// TIA Portal project "template" (V15)

(* hardware
DEVICE "S7-1200 station_1"  S7-1200 Station
   slot 0: "Rack_0"  S7-1200 Rack  Rack  V1.0
   slot 1: "PLC_1"  CPU 1214C AC/DC/Rly  6ES7 214-1BG40-0XB0  V4.2
*)

// ===== PLC "PLC_1"  CPU 1214C AC/DC/Rly =====

VAR_GLOBAL   // PLC tag table "默认变量表"
   "M4.0" AT %M4.0 : Bool;
   "on/off" AT %I0.7 : Bool;
   "start" AT %I0.0 : Bool;
   "M4.1" AT %M4.1 : Bool;
   "water full" AT %I0.1 : Bool;
   "M4.2" AT %M4.2 : Bool;
   "M4.3" AT %M4.3 : Bool;
   "M4.4" AT %M4.4 : Bool;
   "M4.5" AT %M4.5 : Bool;
   "M4.6" AT %M4.6 : Bool;
   "M4.7" AT %M4.7 : Bool;
   "M5.0" AT %M5.0 : Bool;
   "M5.1" AT %M5.1 : Bool;
   "M5.2" AT %M5.2 : Bool;
   "?????????????????" AT %IW30 : Word;
   "cycle of span" AT %MB30 : Byte;
   "cycle of step" AT %MB31 : Byte;
   "water on" AT %Q0.0 : Bool;
   "run+" AT %Q0.1 : Bool;
   "run-" AT %Q0.2 : Bool;
   "tag1" AT %M0.5 : Bool;
   "water off" AT %Q0.3 : Bool;
   "tag2" AT %M0.6 : Bool;
   "water fuck" AT %Q0.4 : Bool;
   "ring" AT %Q0.5 : Bool;
   "stop!!!" AT %I0.2 : Bool;
   "water out" AT %I0.3 : Bool;
   "spanreset" AT %M0.7 : Bool;
   "stepreset" AT %M0.4 : Bool;
END_VAR

// folder: System blocks/Program resources

DATA_BLOCK "IEC_Timer_0_DB"   // DB1
{ S7_Optimized_Access := 'TRUE' }
AUTHOR : Simatic
FAMILY : IEC
NAME : IEC_TMR
VERSION : 1.0
// stored: InstanceOfName IEC_TIMER
"IEC_TIMER"
BEGIN
END_DATA_BLOCK

DATA_BLOCK "IEC_Timer_0_DB_1"   // DB2
{ S7_Optimized_Access := 'TRUE' }
AUTHOR : Simatic
FAMILY : IEC
NAME : IEC_TMR
VERSION : 1.0
// stored: InstanceOfName IEC_TIMER
"IEC_TIMER"
BEGIN
END_DATA_BLOCK

DATA_BLOCK "IEC_Timer_0_DB_2"   // DB3
{ S7_Optimized_Access := 'TRUE' }
AUTHOR : Simatic
FAMILY : IEC
NAME : IEC_TMR
VERSION : 1.0
// stored: InstanceOfName IEC_TIMER
"IEC_TIMER"
BEGIN
END_DATA_BLOCK

DATA_BLOCK "IEC_Timer_0_DB_3"   // DB4
{ S7_Optimized_Access := 'TRUE' }
AUTHOR : Simatic
FAMILY : IEC
NAME : IEC_TMR
VERSION : 1.0
// stored: InstanceOfName IEC_TIMER
"IEC_TIMER"
BEGIN
END_DATA_BLOCK

DATA_BLOCK "IEC_Timer_0_DB_4"   // DB5
{ S7_Optimized_Access := 'TRUE' }
AUTHOR : Simatic
FAMILY : IEC
NAME : IEC_TMR
VERSION : 1.0
// stored: InstanceOfName IEC_TIMER
"IEC_TIMER"
BEGIN
END_DATA_BLOCK

DATA_BLOCK "IEC_Timer_0_DB_5"   // DB6
{ S7_Optimized_Access := 'TRUE' }
AUTHOR : Simatic
FAMILY : IEC
NAME : IEC_TMR
VERSION : 1.0
// stored: InstanceOfName IEC_TIMER
"IEC_TIMER"
BEGIN
END_DATA_BLOCK

DATA_BLOCK "IEC_Timer_0_DB_6"   // DB7
{ S7_Optimized_Access := 'TRUE' }
AUTHOR : Simatic
FAMILY : IEC
NAME : IEC_TMR
VERSION : 1.0
// stored: InstanceOfName IEC_TIMER
"IEC_TIMER"
BEGIN
END_DATA_BLOCK

DATA_BLOCK "IEC_Counter_0_DB"   // DB8
{ S7_Optimized_Access := 'TRUE' }
AUTHOR : Simatic
FAMILY : IEC
NAME : CNTR
VERSION : 1.0
// stored: InstanceOfName IEC_COUNTER
"IEC_COUNTER"
BEGIN
END_DATA_BLOCK

DATA_BLOCK "IEC_Counter_0_DB_1"   // DB9
{ S7_Optimized_Access := 'TRUE' }
AUTHOR : Simatic
FAMILY : IEC
NAME : CNTR
VERSION : 1.0
// stored: InstanceOfName IEC_COUNTER
"IEC_COUNTER"
BEGIN
END_DATA_BLOCK

// folder: (top level)

FUNCTION "STOP" : Void   // FC1, LAD
{ S7_Optimized_Access := 'TRUE' }
VERSION : 0.1
   VAR_INPUT
      "STEP" : Bool;
   END_VAR
BEGIN

REGION Network 1
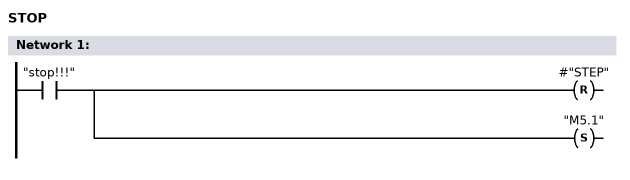
   RUNG wire#powerrail
      Contact( "stop!!!" )
      wire#w1
      R_Coil( #"STEP" )
   END_RUNG
   RUNG wire#w1
      S_Coil( "M5.1" )
   END_RUNG
   // the same network as SCL:
   IF "stop!!!" THEN
       #"STEP" := FALSE;
       "M5.1" := TRUE;
   END_IF;
END_REGION
END_FUNCTION

ORGANIZATION_BLOCK "Main"   // OB1, LAD, ProgramCycle
TITLE = "Main Program Sweep (Cycle)"
{ S7_Optimized_Access := 'TRUE' }
VERSION : 0.1
   VAR_INPUT
      Initial_Call : Bool;   // Initial call of this OB
      Remanence : Bool;   // =True, if remanent data are available
   END_VAR
   VAR_TEMP   // added for the SCL form of the ladder/FBD networks
      _w1 : Bool;
      _w2 : Bool;
      _w3 : Bool;
      _w4 : Bool;
      _w5 : Bool;
      _w6 : Bool;
      _w7 : Bool;
      _w8 : Bool;
      _w9 : Bool;
      _w10 : Bool;
      _w11 : Bool;
      _w12 : Bool;
      _w13 : Bool;
      _w14 : Bool;
      _w15 : Bool;
      _w16 : Bool;
      _w17 : Bool;
      _w18 : Bool;
      _w19 : Bool;
      _w20 : Bool;
   END_VAR
BEGIN

REGION Network 1
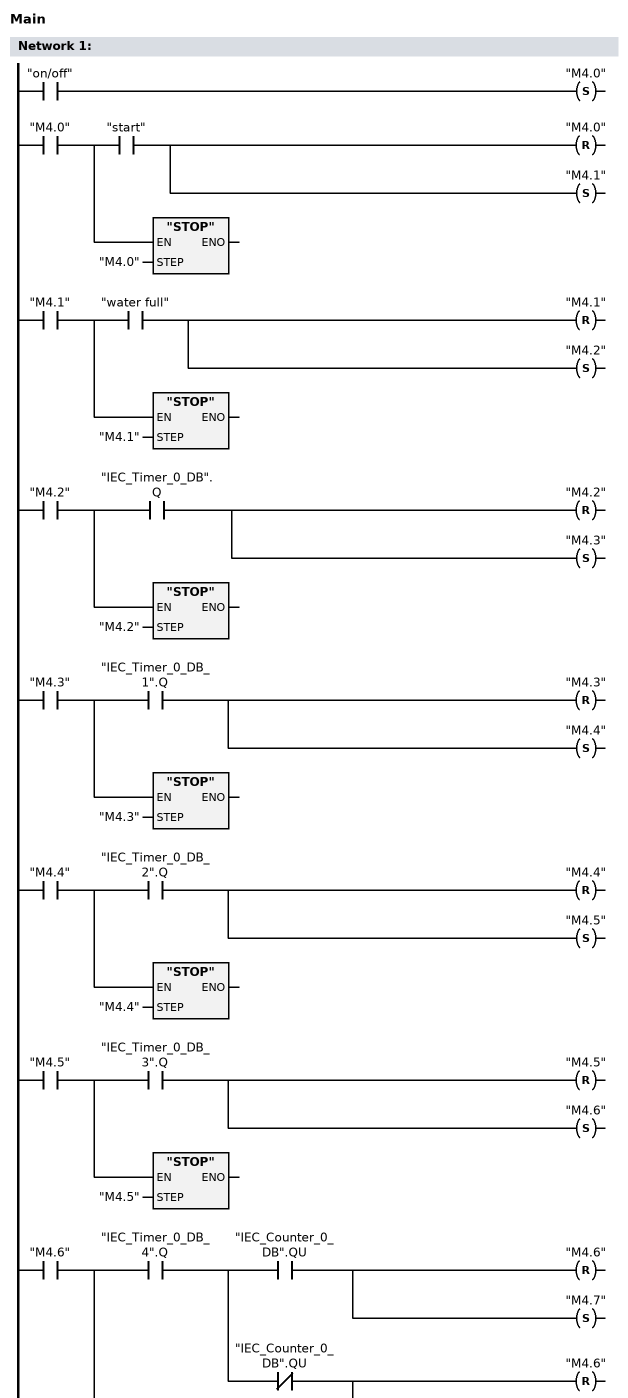
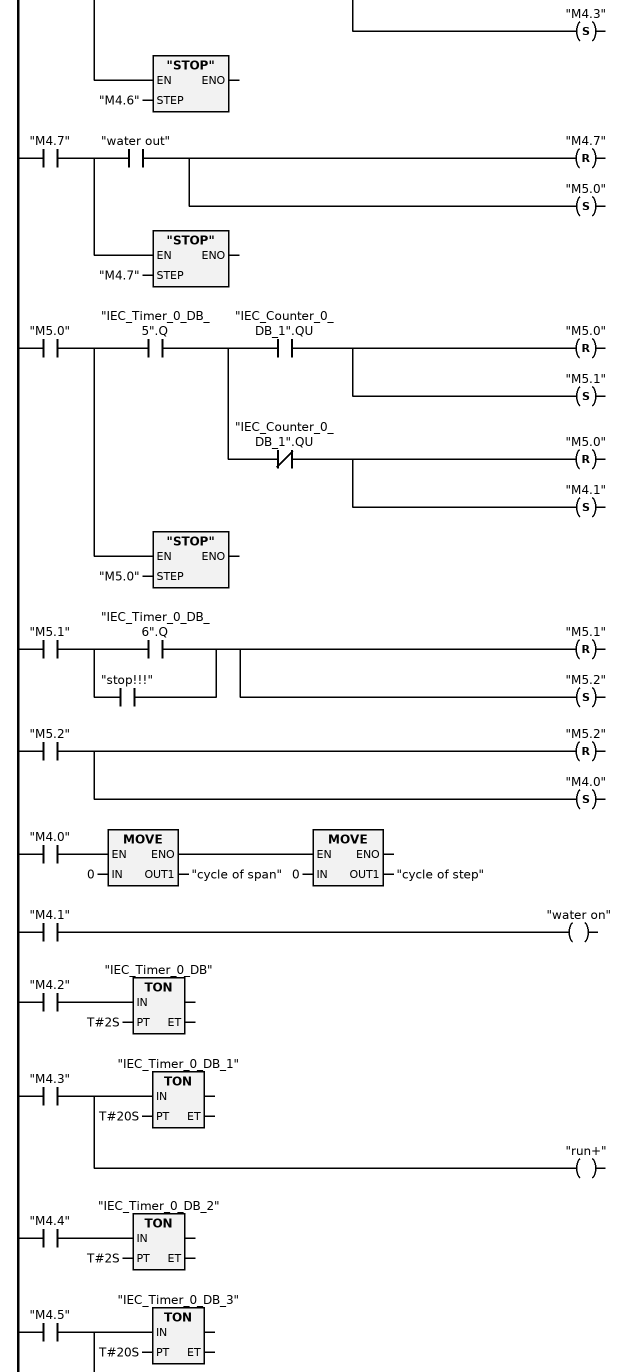
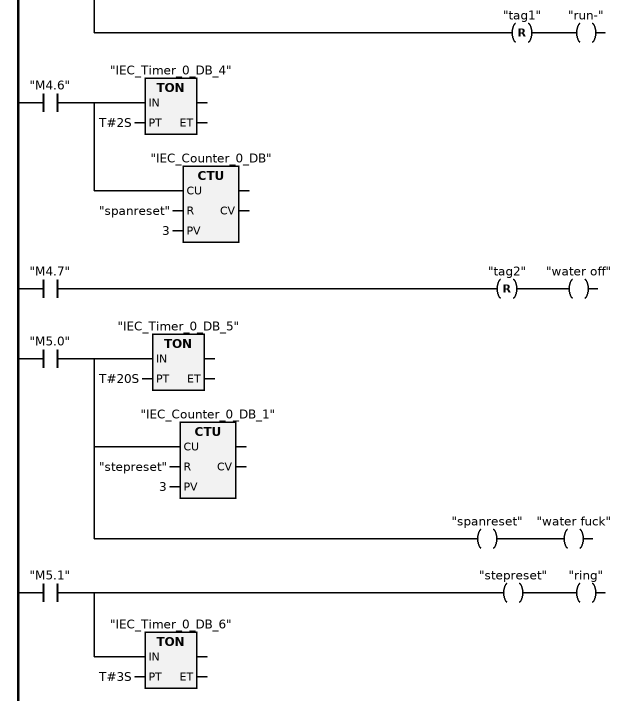
   IF "on/off" THEN "M4.0" := TRUE; END_IF;
   #_w1 := "M4.0";
   #_w2 := "M4.0" AND "start";
   IF #_w2 THEN
       "M4.0" := FALSE;
       "M4.1" := TRUE;
   END_IF;
   IF #_w1 THEN "STOP"("STEP" := "M4.0"); END_IF;
   #_w3 := "M4.1";
   #_w4 := "M4.1" AND "water full";
   IF #_w4 THEN
       "M4.1" := FALSE;
       "M4.2" := TRUE;
   END_IF;
   IF #_w3 THEN "STOP"("STEP" := "M4.1"); END_IF;
   #_w5 := "M4.2";
   #_w6 := "M4.2" AND "IEC_Timer_0_DB".Q;
   IF #_w6 THEN
       "M4.2" := FALSE;
       "M4.3" := TRUE;
   END_IF;
   IF #_w5 THEN "STOP"("STEP" := "M4.2"); END_IF;
   #_w7 := "M4.3";
   #_w8 := "M4.3" AND "IEC_Timer_0_DB_1".Q;
   IF #_w8 THEN
       "M4.3" := FALSE;
       "M4.4" := TRUE;
   END_IF;
   IF #_w7 THEN "STOP"("STEP" := "M4.3"); END_IF;
   #_w9 := "M4.4";
   #_w10 := "M4.4" AND "IEC_Timer_0_DB_2".Q;
   IF #_w10 THEN
       "M4.4" := FALSE;
       "M4.5" := TRUE;
   END_IF;
   IF #_w9 THEN "STOP"("STEP" := "M4.4"); END_IF;
   #_w11 := "M4.5";
   #_w12 := "M4.5" AND "IEC_Timer_0_DB_3".Q;
   IF #_w12 THEN
       "M4.5" := FALSE;
       "M4.6" := TRUE;
   END_IF;
   IF #_w11 THEN "STOP"("STEP" := "M4.5"); END_IF;
   #_w13 := "M4.6" AND "IEC_Timer_0_DB_4".Q;
   #_w14 := "M4.6";
   IF #_w13 AND "IEC_Counter_0_DB".QU THEN
       "M4.6" := FALSE;
       "M4.7" := TRUE;
   END_IF;
   IF #_w13 AND NOT "IEC_Counter_0_DB".QU THEN
       "M4.6" := FALSE;
       "M4.3" := TRUE;
   END_IF;
   IF #_w14 THEN "STOP"("STEP" := "M4.6"); END_IF;
   #_w15 := "M4.7";
   #_w16 := "M4.7" AND "water out";
   IF #_w16 THEN
       "M4.7" := FALSE;
       "M5.0" := TRUE;
   END_IF;
   IF #_w15 THEN "STOP"("STEP" := "M4.7"); END_IF;
   #_w17 := "M5.0" AND "IEC_Timer_0_DB_5".Q;
   #_w18 := "M5.0";
   IF #_w17 AND "IEC_Counter_0_DB_1".QU THEN
       "M5.0" := FALSE;
       "M5.1" := TRUE;
   END_IF;
   IF #_w17 AND NOT "IEC_Counter_0_DB_1".QU THEN
       "M5.0" := FALSE;
       "M4.1" := TRUE;
   END_IF;
   IF #_w18 THEN "STOP"("STEP" := "M5.0"); END_IF;
   #_w19 := "M5.1" AND ("IEC_Timer_0_DB_6".Q OR "stop!!!");
   IF #_w19 THEN
       "M5.1" := FALSE;
       "M5.2" := TRUE;
   END_IF;
   #_w20 := "M5.2";
   IF #_w20 THEN
       "M5.2" := FALSE;
       "M4.0" := TRUE;
   END_IF;
   IF "M4.0" THEN
       "cycle of span" := 0;
       "cycle of step" := 0;
   END_IF;
   "water on" := "M4.1";
   "IEC_Timer_0_DB".TON(IN := "M4.2", PT := T#2S);
   "IEC_Timer_0_DB_1".TON(IN := "M4.3", PT := T#20S);
   "run+" := "M4.3";
   "IEC_Timer_0_DB_2".TON(IN := "M4.4", PT := T#2S);
   "IEC_Timer_0_DB_3".TON(IN := "M4.5", PT := T#20S);
   IF "M4.5" THEN "tag1" := FALSE; END_IF;
   "run-" := "M4.5";
   "IEC_Timer_0_DB_4".TON(IN := "M4.6", PT := T#2S);
   "IEC_Counter_0_DB".CTU(CU := "M4.6", R := "spanreset", PV := 3);
   IF "M4.7" THEN "tag2" := FALSE; END_IF;
   "water off" := "M4.7";
   "IEC_Timer_0_DB_5".TON(IN := "M5.0", PT := T#20S);
   "IEC_Counter_0_DB_1".CTU(CU := "M5.0", R := "stepreset", PV := 3);
   "spanreset" := "M5.0";
   "water fuck" := "M5.0";
   "stepreset" := "M5.1";
   "ring" := "M5.1";
   "IEC_Timer_0_DB_6".TON(IN := "M5.1", PT := T#3S);
END_REGION
END_ORGANIZATION_BLOCK